Universal Robots PolyScope program: reciprocal_p1_2.urp

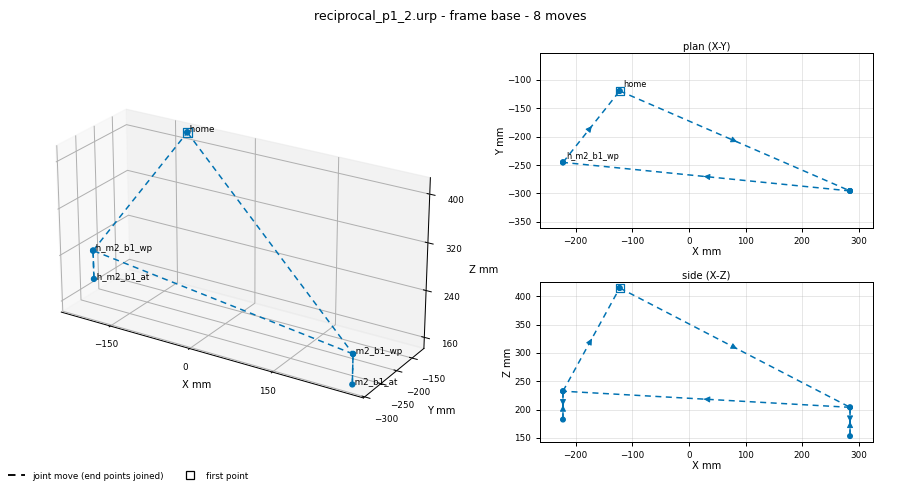
[picture p0: tool path of reciprocal_p1_2.urp in frame base, 8 of 8 moves have a stored position in this frame; points joined in program order, loops and branches not executed]
Program reciprocal_p1_2 (installation=default directory=/programs/usbdisk/ITER createdIn=5.3.1.64192 lastSavedIn=5.3.1.64192 robotSerialNumber=20195300365)
Calibrated DH parameters: a=[-0.000093, -0.190649, -0.212673, 0.000091, -0.000205, 0]; d=[0.151591, 44.061648, -42.488068, -1.442789, 0.085322, 0.091911]; alpha=[1.570082, -0.003447, 0.007513, 1.572293, -1.571904, 0]; deltaTheta=[0, -0.672656, 0.728185, -0.055522, 0.000005, 0]
Robot Program (runOnlyOnce=false)
  URCap Gripper Activate (Robotiq_Grippers, Robotiq Inc.) dataModel(ResetAndActivateKey=false)
  URCap Gripper (Robotiq_Grippers, Robotiq Inc.) dataModel(position=50.0, force=100.0, speed=100.0, positionInDouble=50.0, forceInDouble=100.0, speedInDouble=100.0, slaveIds=[9], blocking=true)
  MoveJ speed 60 deg/s, acceleration 80 deg/s^2 (useActiveTCP=true) feature=Base
    Waypoint home: TCP in base x=-122.15 y=-119.32 z=414.454 mm, rx=2.2563 ry=2.1459 rz=-0.0481 rad; joints [-85.681, -56.776, -79.802, -131.025, 89.944, -262.833] deg
  Folder Mid_2
    MoveJ speed 60 deg/s, acceleration 80 deg/s^2 (useActiveTCP=true) feature=Base
      Waypoint m2_b1_wp: TCP in base x=284.16 y=-295.685 z=203.947 mm, rx=2.2476 ry=2.1381 rz=-0.0269 rad; joints [-27.296, -114.823, -87.386, -65.934, 88.586, -204.141] deg
      Waypoint m2_b1_at: TCP in base x=284.146 y=-295.69 z=153.108 mm, rx=2.2477 ry=2.1381 rz=-0.0269 rad; joints [-27.314, -120.451, -93.885, -53.812, 88.539, -204.094] deg
      URCap Gripper (Robotiq_Grippers, Robotiq Inc.) dataModel(position=100.0, force=100.0, speed=100.0, positionInDouble=100.0, forceInDouble=100.0, speedInDouble=100.0, slaveIds=[9], blocking=true)
      Waypoint m2_b1_wp: TCP in base x=284.16 y=-295.685 z=203.947 mm, rx=2.2476 ry=2.1381 rz=-0.0269 rad; joints [-27.296, -114.823, -87.386, -65.934, 88.586, -204.141] deg
      Waypoint h_m2_b1_wp: TCP in base x=-222.193 y=-245.34 z=232.403 mm, rx=-3.1314 ry=0.0205 rz=0.0123 rad; joints [-108.936, -94.247, -105.13, -70.966, 89.712, -197.837] deg
      Waypoint h_m2_b1_at: TCP in base x=-222.194 y=-245.343 z=182.32 mm, rx=-3.1314 ry=0.0205 rz=0.0122 rad; joints [-108.96, -99.771, -113.792, -56.782, 89.658, -197.776] deg
      URCap Gripper (Robotiq_Grippers, Robotiq Inc.) dataModel(position=50.0, force=100.0, speed=100.0, positionInDouble=50.0, forceInDouble=100.0, speedInDouble=100.0, slaveIds=[9], blocking=true)
      Waypoint h_m2_b1_wp: TCP in base x=-222.193 y=-245.34 z=232.403 mm, rx=-3.1314 ry=0.0205 rz=0.0123 rad; joints [-108.936, -94.247, -105.13, -70.966, 89.712, -197.837] deg
  MoveJ speed 60 deg/s, acceleration 80 deg/s^2 (useActiveTCP=true) feature=Base
    Waypoint home: TCP in base x=-122.15 y=-119.32 z=414.454 mm, rx=2.2563 ry=2.1459 rz=-0.0481 rad; joints [-85.681, -56.776, -79.802, -131.025, 89.944, -262.833] deg
